// TIA Portal V19 export
DATA_BLOCK "CallEquipmentMotionCycle_DB"   // DB176
{ DB_Accessible_From_OPC_UA := 'FALSE' }
// stored: DBAccessibleFromOPCUA false, DBAccessibleFromWebserver false, InstanceOfName Unit.Em2.CallEquipmentMotionCycle, InstanceOfType FB, Namespace Unit.Em2
"Unit.Em2.CallEquipmentMotionCycle"
   // VAR_OUTPUT
   //    error { ExternalAccessible := 'False'; ExternalVisible := 'False'; ExternalWritable := 'False'} : Bool;
   // END_VAR
   // VAR_IN_OUT
   //    syncNode : "Unit.Em2.typeSyncNode";
   // END_VAR
BEGIN
END_DATA_BLOCK
